PROGRAM main
VAR
END_VAR

// Main function for testing some functionality

testShelf();

// testFlexiBuffer();

END_PROGRAM

(* stored: Version 1.1.0.1
   POU main: Id {a5da58b8-5a34-42e4-a5de-1b0ec0c09d5b}, SpecialFunc None *)
